{attribute 'qualified_only'}
VAR_GLOBAL
END_VAR

(* stored: Version 1.1.0.1, ProductVersion 3.1.4022.7
   GVL GVL_05_Manual_Servo_Motor_Shelf_C: Id {a62afa05-e243-4404-8c90-5bea922d5bfc} *)
